PROGRAM P3_05_BatchTrail
VAR
	stDBParam 					:ST_BatchTrail;	
	fbDBWrite					:FB_PLCDBWriteEvt(sNetId:=CONST.AMS_NETID, tTimeout:=DEFAULT_ADS_TIMEOUT);
	tableColumns				:ARRAY [0..5] OF STRING(50) := ['batch', 'event', 'description', 'user', 'oldvalue', 'newvalue'];
	arrParam					:ARRAY [0..5] OF ST_ExpParameter := [(sParaName := 'batch', nParaSize := 101, eParaType := E_EXPPARAMETERTYPE.STRING_),
															 (sParaName := 'event', nParaSize := 101, eParaType := E_EXPPARAMETERTYPE.STRING_),
															 (sParaName := 'description', nParaSize := 101, eParaType := E_EXPPARAMETERTYPE.STRING_),
															 (sParaName := 'user', nParaSize := 101, eParaType := E_EXPPARAMETERTYPE.STRING_),
															 (sParaName := 'oldvalue', nParaSize := 101, eParaType := E_EXPPARAMETERTYPE.STRING_),
															 (sParaName := 'newvalue', nParaSize := 101, eParaType := E_EXPPARAMETERTYPE.STRING_)];
	fbDeleteTable    			:FB_PLCDBCmdEvt(sNetID:=CONST.AMS_NETID, tTimeout:=DEFAULT_ADS_TIMEOUT);
	fbBatchTrailWrite			:ARRAY[0..70] OF FB_AuditTrail_Write;
	sDeleteBatch				:STRING;	
	sDeleteAll					:STRING;
	sDelete						:STRING;
	bDelete						:BOOL;								
	bWrite						:BOOL;
	
	sProdCurrentPhase			:STRING;
	sCleanCurrentPhase			:STRING;
END_VAR
VAR // added by the converter: edge detectors and wires of the graphical bodies
    _rt1 : R_TRIG;
END_VAR

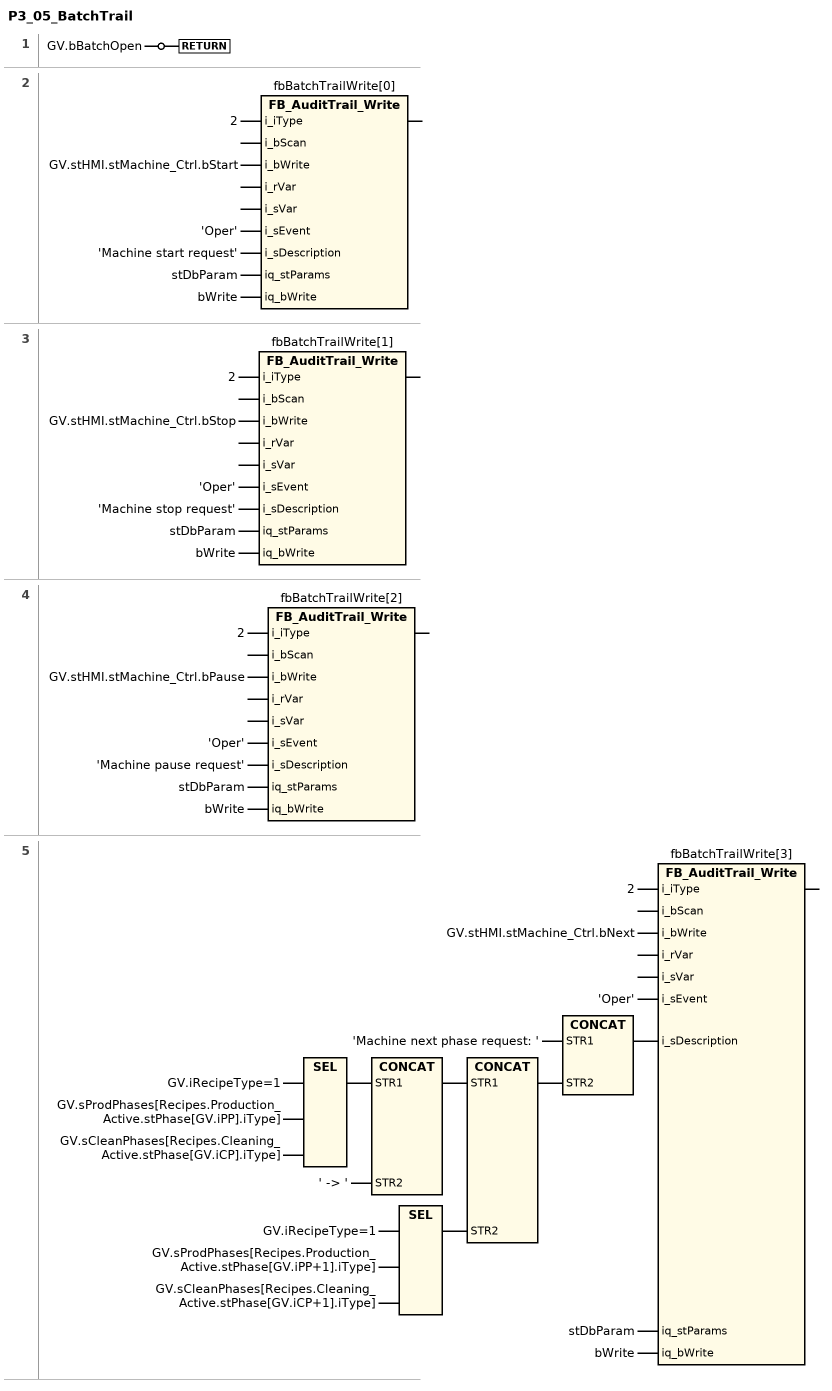
// NETWORK 1
IF NOT GV.bBatchOpen THEN RETURN; END_IF

// NETWORK 2
fbBatchTrailWrite[0](
    i_iType := 2,
    i_bWrite := GV.stHMI.stMachine_Ctrl.bStart,
    i_sEvent := 'Oper',
    i_sDescription := 'Machine start request',
    iq_stParams := stDbParam,
    iq_bWrite := bWrite); // FB_AuditTrail_Write

// NETWORK 3
fbBatchTrailWrite[1](
    i_iType := 2,
    i_bWrite := GV.stHMI.stMachine_Ctrl.bStop,
    i_sEvent := 'Oper',
    i_sDescription := 'Machine stop request',
    iq_stParams := stDbParam,
    iq_bWrite := bWrite); // FB_AuditTrail_Write

// NETWORK 4
fbBatchTrailWrite[2](
    i_iType := 2,
    i_bWrite := GV.stHMI.stMachine_Ctrl.bPause,
    i_sEvent := 'Oper',
    i_sDescription := 'Machine pause request',
    iq_stParams := stDbParam,
    iq_bWrite := bWrite); // FB_AuditTrail_Write

// NETWORK 5
fbBatchTrailWrite[3](
    i_iType := 2,
    i_bWrite := GV.stHMI.stMachine_Ctrl.bNext,
    i_sEvent := 'Oper',
    i_sDescription := CONCAT(STR1 := 'Machine next phase request: ', STR2 := CONCAT(STR1 := CONCAT(STR1 := SEL(GV.iRecipeType=1, GV.sProdPhases[Recipes.Production_Active.stPhase[GV.iPP].iType], GV.sCleanPhases[Recipes.Cleaning_Active.stPhase[GV.iCP].iType]), STR2 := ' -> '), STR2 := SEL(GV.iRecipeType=1, GV.sProdPhases[Recipes.Production_Active.stPhase[GV.iPP+1].iType], GV.sCleanPhases[Recipes.Cleaning_Active.stPhase[GV.iCP+1].iType]))),
    iq_stParams := stDbParam,
    iq_bWrite := bWrite); // FB_AuditTrail_Write

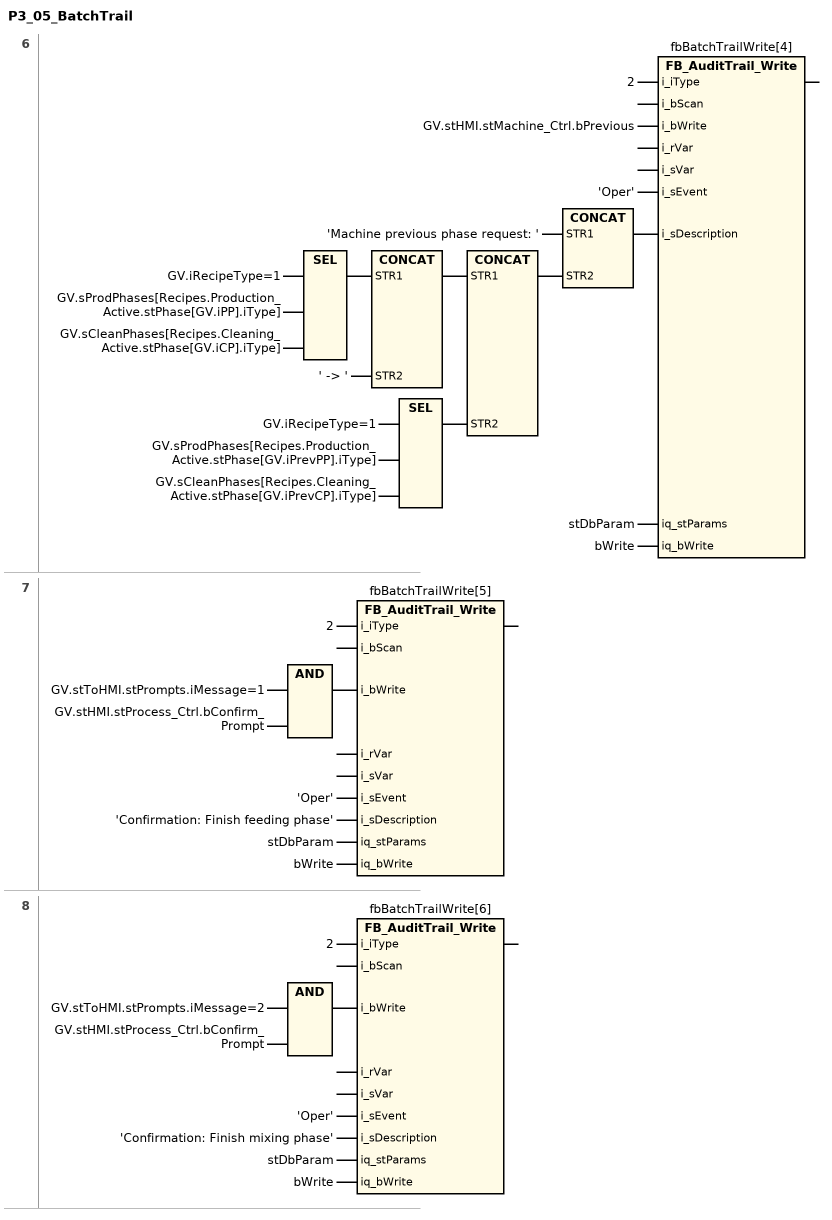
// NETWORK 6
fbBatchTrailWrite[4](
    i_iType := 2,
    i_bWrite := GV.stHMI.stMachine_Ctrl.bPrevious,
    i_sEvent := 'Oper',
    i_sDescription := CONCAT(STR1 := 'Machine previous phase request: ', STR2 := CONCAT(STR1 := CONCAT(STR1 := SEL(GV.iRecipeType=1, GV.sProdPhases[Recipes.Production_Active.stPhase[GV.iPP].iType], GV.sCleanPhases[Recipes.Cleaning_Active.stPhase[GV.iCP].iType]), STR2 := ' -> '), STR2 := SEL(GV.iRecipeType=1, GV.sProdPhases[Recipes.Production_Active.stPhase[GV.iPrevPP].iType], GV.sCleanPhases[Recipes.Cleaning_Active.stPhase[GV.iPrevCP].iType]))),
    iq_stParams := stDbParam,
    iq_bWrite := bWrite); // FB_AuditTrail_Write

// NETWORK 7
fbBatchTrailWrite[5](
    i_iType := 2,
    i_bWrite := (GV.stToHMI.stPrompts.iMessage=1) AND GV.stHMI.stProcess_Ctrl.bConfirm_Prompt,
    i_sEvent := 'Oper',
    i_sDescription := 'Confirmation: Finish feeding phase',
    iq_stParams := stDbParam,
    iq_bWrite := bWrite); // FB_AuditTrail_Write

// NETWORK 8
fbBatchTrailWrite[6](
    i_iType := 2,
    i_bWrite := (GV.stToHMI.stPrompts.iMessage=2) AND GV.stHMI.stProcess_Ctrl.bConfirm_Prompt,
    i_sEvent := 'Oper',
    i_sDescription := 'Confirmation: Finish mixing phase',
    iq_stParams := stDbParam,
    iq_bWrite := bWrite); // FB_AuditTrail_Write

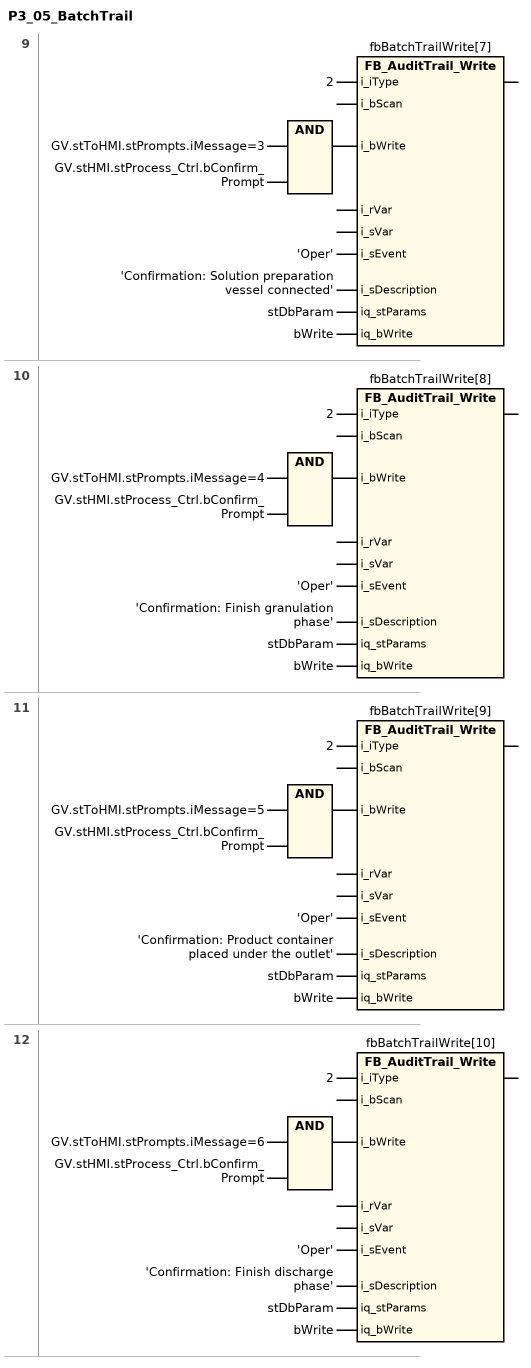
// NETWORK 9
fbBatchTrailWrite[7](
    i_iType := 2,
    i_bWrite := (GV.stToHMI.stPrompts.iMessage=3) AND GV.stHMI.stProcess_Ctrl.bConfirm_Prompt,
    i_sEvent := 'Oper',
    i_sDescription := 'Confirmation: Solution preparation vessel connected',
    iq_stParams := stDbParam,
    iq_bWrite := bWrite); // FB_AuditTrail_Write

// NETWORK 10
fbBatchTrailWrite[8](
    i_iType := 2,
    i_bWrite := (GV.stToHMI.stPrompts.iMessage=4) AND GV.stHMI.stProcess_Ctrl.bConfirm_Prompt,
    i_sEvent := 'Oper',
    i_sDescription := 'Confirmation: Finish granulation phase',
    iq_stParams := stDbParam,
    iq_bWrite := bWrite); // FB_AuditTrail_Write

// NETWORK 11
fbBatchTrailWrite[9](
    i_iType := 2,
    i_bWrite := (GV.stToHMI.stPrompts.iMessage=5) AND GV.stHMI.stProcess_Ctrl.bConfirm_Prompt,
    i_sEvent := 'Oper',
    i_sDescription := 'Confirmation: Product container placed under the outlet',
    iq_stParams := stDbParam,
    iq_bWrite := bWrite); // FB_AuditTrail_Write

// NETWORK 12
fbBatchTrailWrite[10](
    i_iType := 2,
    i_bWrite := (GV.stToHMI.stPrompts.iMessage=6) AND GV.stHMI.stProcess_Ctrl.bConfirm_Prompt,
    i_sEvent := 'Oper',
    i_sDescription := 'Confirmation: Finish discharge phase',
    iq_stParams := stDbParam,
    iq_bWrite := bWrite); // FB_AuditTrail_Write

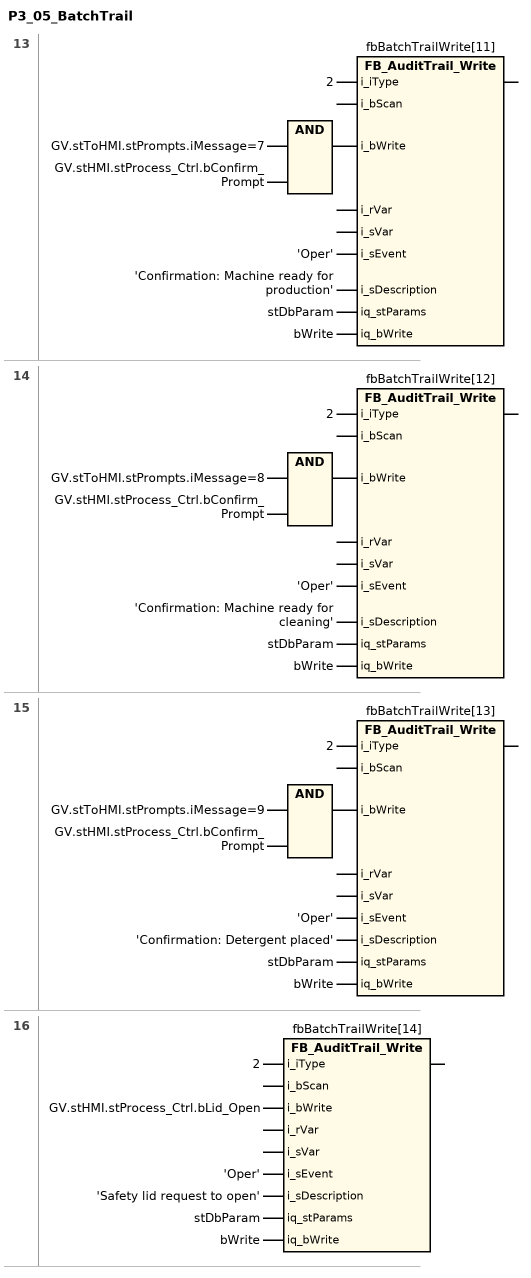
// NETWORK 13
fbBatchTrailWrite[11](
    i_iType := 2,
    i_bWrite := (GV.stToHMI.stPrompts.iMessage=7) AND GV.stHMI.stProcess_Ctrl.bConfirm_Prompt,
    i_sEvent := 'Oper',
    i_sDescription := 'Confirmation: Machine ready for production',
    iq_stParams := stDbParam,
    iq_bWrite := bWrite); // FB_AuditTrail_Write

// NETWORK 14
fbBatchTrailWrite[12](
    i_iType := 2,
    i_bWrite := (GV.stToHMI.stPrompts.iMessage=8) AND GV.stHMI.stProcess_Ctrl.bConfirm_Prompt,
    i_sEvent := 'Oper',
    i_sDescription := 'Confirmation: Machine ready for cleaning',
    iq_stParams := stDbParam,
    iq_bWrite := bWrite); // FB_AuditTrail_Write

// NETWORK 15
fbBatchTrailWrite[13](
    i_iType := 2,
    i_bWrite := (GV.stToHMI.stPrompts.iMessage=9) AND GV.stHMI.stProcess_Ctrl.bConfirm_Prompt,
    i_sEvent := 'Oper',
    i_sDescription := 'Confirmation: Detergent placed',
    iq_stParams := stDbParam,
    iq_bWrite := bWrite); // FB_AuditTrail_Write

// NETWORK 16
fbBatchTrailWrite[14](
    i_iType := 2,
    i_bWrite := GV.stHMI.stProcess_Ctrl.bLid_Open,
    i_sEvent := 'Oper',
    i_sDescription := 'Safety lid request to open',
    iq_stParams := stDbParam,
    iq_bWrite := bWrite); // FB_AuditTrail_Write

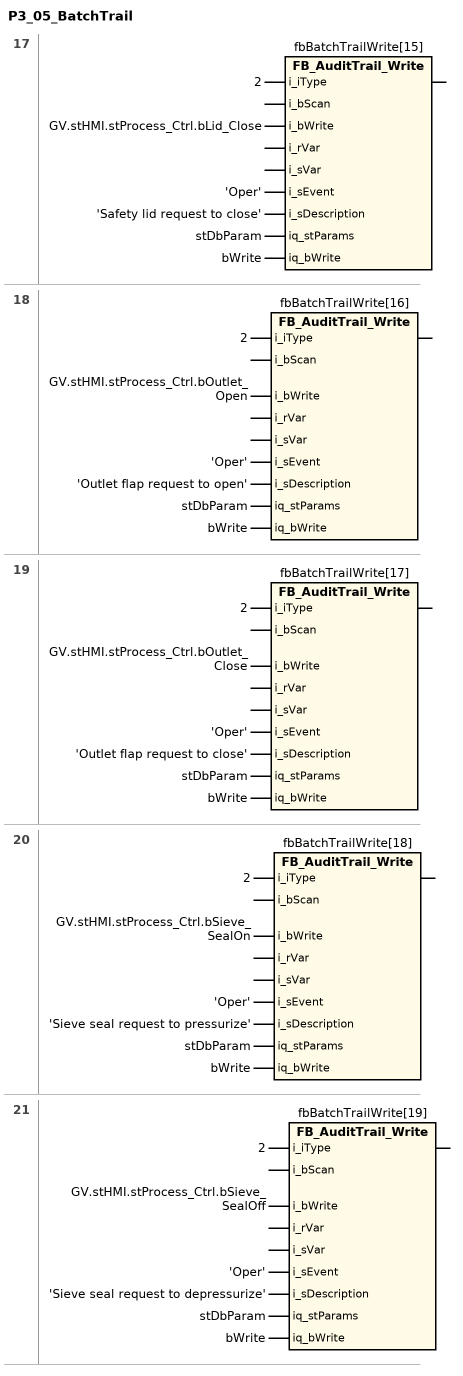
// NETWORK 17
fbBatchTrailWrite[15](
    i_iType := 2,
    i_bWrite := GV.stHMI.stProcess_Ctrl.bLid_Close,
    i_sEvent := 'Oper',
    i_sDescription := 'Safety lid request to close',
    iq_stParams := stDbParam,
    iq_bWrite := bWrite); // FB_AuditTrail_Write

// NETWORK 18
fbBatchTrailWrite[16](
    i_iType := 2,
    i_bWrite := GV.stHMI.stProcess_Ctrl.bOutlet_Open,
    i_sEvent := 'Oper',
    i_sDescription := 'Outlet flap request to open',
    iq_stParams := stDbParam,
    iq_bWrite := bWrite); // FB_AuditTrail_Write

// NETWORK 19
fbBatchTrailWrite[17](
    i_iType := 2,
    i_bWrite := GV.stHMI.stProcess_Ctrl.bOutlet_Close,
    i_sEvent := 'Oper',
    i_sDescription := 'Outlet flap request to close',
    iq_stParams := stDbParam,
    iq_bWrite := bWrite); // FB_AuditTrail_Write

// NETWORK 20
fbBatchTrailWrite[18](
    i_iType := 2,
    i_bWrite := GV.stHMI.stProcess_Ctrl.bSieve_SealOn,
    i_sEvent := 'Oper',
    i_sDescription := 'Sieve seal request to pressurize',
    iq_stParams := stDbParam,
    iq_bWrite := bWrite); // FB_AuditTrail_Write

// NETWORK 21
fbBatchTrailWrite[19](
    i_iType := 2,
    i_bWrite := GV.stHMI.stProcess_Ctrl.bSieve_SealOff,
    i_sEvent := 'Oper',
    i_sDescription := 'Sieve seal request to depressurize',
    iq_stParams := stDbParam,
    iq_bWrite := bWrite); // FB_AuditTrail_Write

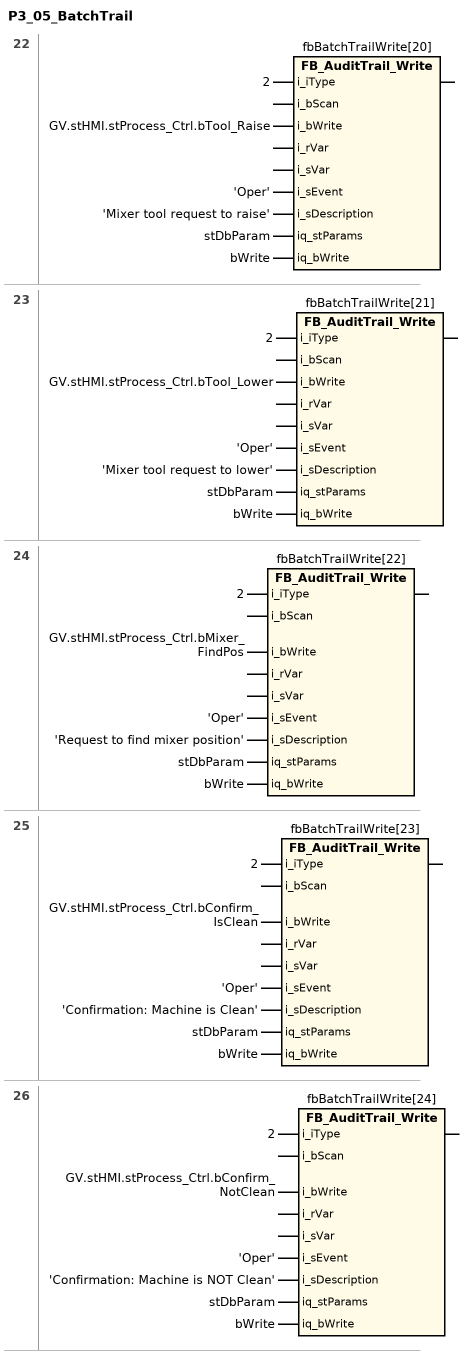
// NETWORK 22
fbBatchTrailWrite[20](
    i_iType := 2,
    i_bWrite := GV.stHMI.stProcess_Ctrl.bTool_Raise,
    i_sEvent := 'Oper',
    i_sDescription := 'Mixer tool request to raise',
    iq_stParams := stDbParam,
    iq_bWrite := bWrite); // FB_AuditTrail_Write

// NETWORK 23
fbBatchTrailWrite[21](
    i_iType := 2,
    i_bWrite := GV.stHMI.stProcess_Ctrl.bTool_Lower,
    i_sEvent := 'Oper',
    i_sDescription := 'Mixer tool request to lower',
    iq_stParams := stDbParam,
    iq_bWrite := bWrite); // FB_AuditTrail_Write

// NETWORK 24
fbBatchTrailWrite[22](
    i_iType := 2,
    i_bWrite := GV.stHMI.stProcess_Ctrl.bMixer_FindPos,
    i_sEvent := 'Oper',
    i_sDescription := 'Request to find mixer position',
    iq_stParams := stDbParam,
    iq_bWrite := bWrite); // FB_AuditTrail_Write

// NETWORK 25
fbBatchTrailWrite[23](
    i_iType := 2,
    i_bWrite := GV.stHMI.stProcess_Ctrl.bConfirm_IsClean,
    i_sEvent := 'Oper',
    i_sDescription := 'Confirmation: Machine is Clean',
    iq_stParams := stDbParam,
    iq_bWrite := bWrite); // FB_AuditTrail_Write

// NETWORK 26
fbBatchTrailWrite[24](
    i_iType := 2,
    i_bWrite := GV.stHMI.stProcess_Ctrl.bConfirm_NotClean,
    i_sEvent := 'Oper',
    i_sDescription := 'Confirmation: Machine is NOT Clean',
    iq_stParams := stDbParam,
    iq_bWrite := bWrite); // FB_AuditTrail_Write

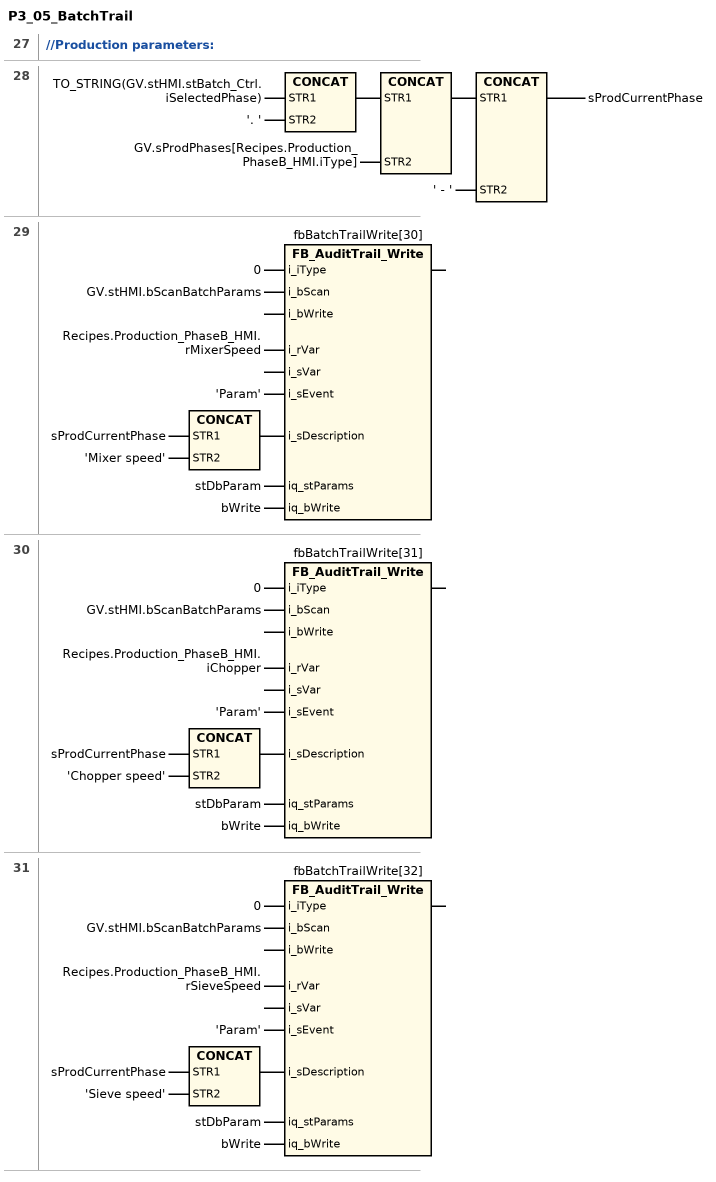
// NETWORK 27
// label: //Production parameters

// NETWORK 28
sProdCurrentPhase := CONCAT(STR1 := CONCAT(STR1 := CONCAT(STR1 := TO_STRING(GV.stHMI.stBatch_Ctrl.iSelectedPhase), STR2 := '. '), STR2 := GV.sProdPhases[Recipes.Production_PhaseB_HMI.iType]), STR2 := ' - ');

// NETWORK 29
fbBatchTrailWrite[30](
    i_iType := 0,
    i_bScan := GV.stHMI.bScanBatchParams,
    i_rVar := Recipes.Production_PhaseB_HMI.rMixerSpeed,
    i_sEvent := 'Param',
    i_sDescription := CONCAT(STR1 := sProdCurrentPhase, STR2 := 'Mixer speed'),
    iq_stParams := stDbParam,
    iq_bWrite := bWrite); // FB_AuditTrail_Write

// NETWORK 30
fbBatchTrailWrite[31](
    i_iType := 0,
    i_bScan := GV.stHMI.bScanBatchParams,
    i_rVar := Recipes.Production_PhaseB_HMI.iChopper,
    i_sEvent := 'Param',
    i_sDescription := CONCAT(STR1 := sProdCurrentPhase, STR2 := 'Chopper speed'),
    iq_stParams := stDbParam,
    iq_bWrite := bWrite); // FB_AuditTrail_Write

// NETWORK 31
fbBatchTrailWrite[32](
    i_iType := 0,
    i_bScan := GV.stHMI.bScanBatchParams,
    i_rVar := Recipes.Production_PhaseB_HMI.rSieveSpeed,
    i_sEvent := 'Param',
    i_sDescription := CONCAT(STR1 := sProdCurrentPhase, STR2 := 'Sieve speed'),
    iq_stParams := stDbParam,
    iq_bWrite := bWrite); // FB_AuditTrail_Write

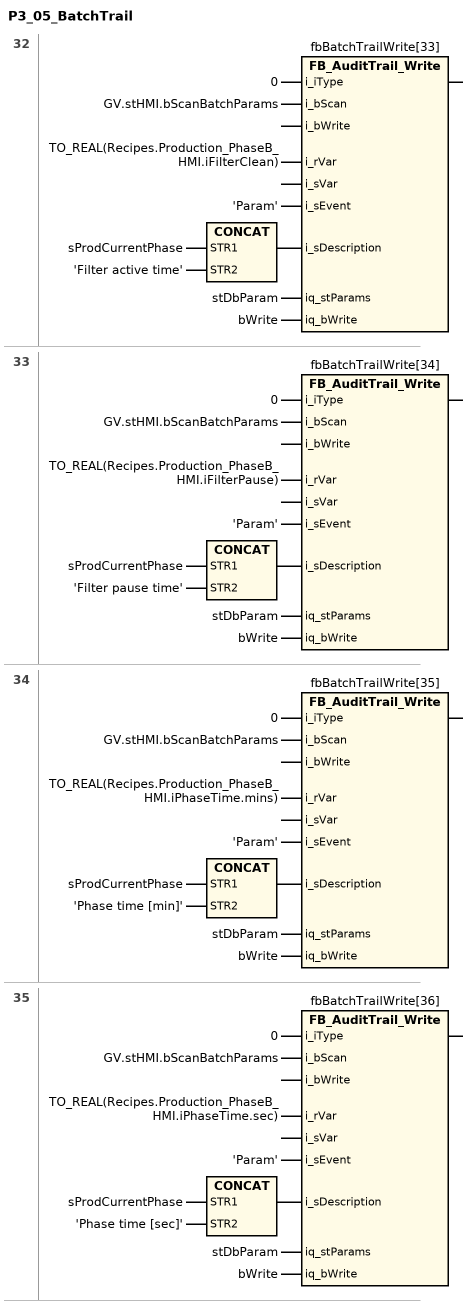
// NETWORK 32
fbBatchTrailWrite[33](
    i_iType := 0,
    i_bScan := GV.stHMI.bScanBatchParams,
    i_rVar := TO_REAL(Recipes.Production_PhaseB_HMI.iFilterClean),
    i_sEvent := 'Param',
    i_sDescription := CONCAT(STR1 := sProdCurrentPhase, STR2 := 'Filter active time'),
    iq_stParams := stDbParam,
    iq_bWrite := bWrite); // FB_AuditTrail_Write

// NETWORK 33
fbBatchTrailWrite[34](
    i_iType := 0,
    i_bScan := GV.stHMI.bScanBatchParams,
    i_rVar := TO_REAL(Recipes.Production_PhaseB_HMI.iFilterPause),
    i_sEvent := 'Param',
    i_sDescription := CONCAT(STR1 := sProdCurrentPhase, STR2 := 'Filter pause time'),
    iq_stParams := stDbParam,
    iq_bWrite := bWrite); // FB_AuditTrail_Write

// NETWORK 34
fbBatchTrailWrite[35](
    i_iType := 0,
    i_bScan := GV.stHMI.bScanBatchParams,
    i_rVar := TO_REAL(Recipes.Production_PhaseB_HMI.iPhaseTime.mins),
    i_sEvent := 'Param',
    i_sDescription := CONCAT(STR1 := sProdCurrentPhase, STR2 := 'Phase time [min]'),
    iq_stParams := stDbParam,
    iq_bWrite := bWrite); // FB_AuditTrail_Write

// NETWORK 35
fbBatchTrailWrite[36](
    i_iType := 0,
    i_bScan := GV.stHMI.bScanBatchParams,
    i_rVar := TO_REAL(Recipes.Production_PhaseB_HMI.iPhaseTime.sec),
    i_sEvent := 'Param',
    i_sDescription := CONCAT(STR1 := sProdCurrentPhase, STR2 := 'Phase time [sec]'),
    iq_stParams := stDbParam,
    iq_bWrite := bWrite); // FB_AuditTrail_Write

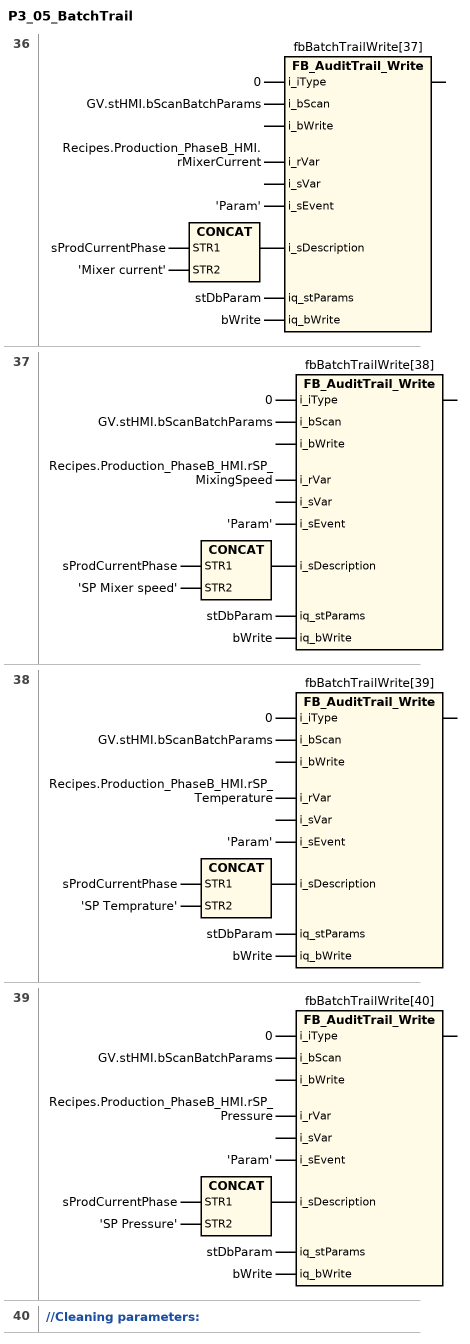
// NETWORK 36
fbBatchTrailWrite[37](
    i_iType := 0,
    i_bScan := GV.stHMI.bScanBatchParams,
    i_rVar := Recipes.Production_PhaseB_HMI.rMixerCurrent,
    i_sEvent := 'Param',
    i_sDescription := CONCAT(STR1 := sProdCurrentPhase, STR2 := 'Mixer current'),
    iq_stParams := stDbParam,
    iq_bWrite := bWrite); // FB_AuditTrail_Write

// NETWORK 37
fbBatchTrailWrite[38](
    i_iType := 0,
    i_bScan := GV.stHMI.bScanBatchParams,
    i_rVar := Recipes.Production_PhaseB_HMI.rSP_MixingSpeed,
    i_sEvent := 'Param',
    i_sDescription := CONCAT(STR1 := sProdCurrentPhase, STR2 := 'SP Mixer speed'),
    iq_stParams := stDbParam,
    iq_bWrite := bWrite); // FB_AuditTrail_Write

// NETWORK 38
fbBatchTrailWrite[39](
    i_iType := 0,
    i_bScan := GV.stHMI.bScanBatchParams,
    i_rVar := Recipes.Production_PhaseB_HMI.rSP_Temperature,
    i_sEvent := 'Param',
    i_sDescription := CONCAT(STR1 := sProdCurrentPhase, STR2 := 'SP Temprature'),
    iq_stParams := stDbParam,
    iq_bWrite := bWrite); // FB_AuditTrail_Write

// NETWORK 39
fbBatchTrailWrite[40](
    i_iType := 0,
    i_bScan := GV.stHMI.bScanBatchParams,
    i_rVar := Recipes.Production_PhaseB_HMI.rSP_Pressure,
    i_sEvent := 'Param',
    i_sDescription := CONCAT(STR1 := sProdCurrentPhase, STR2 := 'SP Pressure'),
    iq_stParams := stDbParam,
    iq_bWrite := bWrite); // FB_AuditTrail_Write

// NETWORK 40
// label: //Cleaning parameters

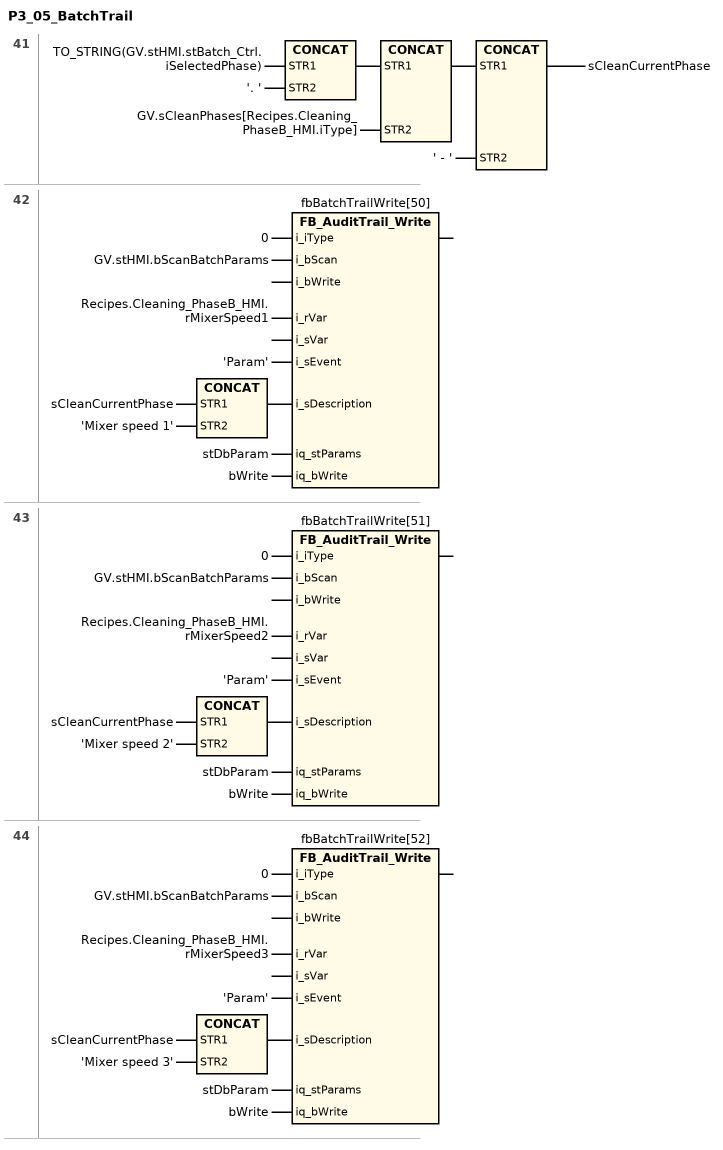
// NETWORK 41
sCleanCurrentPhase := CONCAT(STR1 := CONCAT(STR1 := CONCAT(STR1 := TO_STRING(GV.stHMI.stBatch_Ctrl.iSelectedPhase), STR2 := '. '), STR2 := GV.sCleanPhases[Recipes.Cleaning_PhaseB_HMI.iType]), STR2 := ' - ');

// NETWORK 42
fbBatchTrailWrite[50](
    i_iType := 0,
    i_bScan := GV.stHMI.bScanBatchParams,
    i_rVar := Recipes.Cleaning_PhaseB_HMI.rMixerSpeed1,
    i_sEvent := 'Param',
    i_sDescription := CONCAT(STR1 := sCleanCurrentPhase, STR2 := 'Mixer speed 1'),
    iq_stParams := stDbParam,
    iq_bWrite := bWrite); // FB_AuditTrail_Write

// NETWORK 43
fbBatchTrailWrite[51](
    i_iType := 0,
    i_bScan := GV.stHMI.bScanBatchParams,
    i_rVar := Recipes.Cleaning_PhaseB_HMI.rMixerSpeed2,
    i_sEvent := 'Param',
    i_sDescription := CONCAT(STR1 := sCleanCurrentPhase, STR2 := 'Mixer speed 2'),
    iq_stParams := stDbParam,
    iq_bWrite := bWrite); // FB_AuditTrail_Write

// NETWORK 44
fbBatchTrailWrite[52](
    i_iType := 0,
    i_bScan := GV.stHMI.bScanBatchParams,
    i_rVar := Recipes.Cleaning_PhaseB_HMI.rMixerSpeed3,
    i_sEvent := 'Param',
    i_sDescription := CONCAT(STR1 := sCleanCurrentPhase, STR2 := 'Mixer speed 3'),
    iq_stParams := stDbParam,
    iq_bWrite := bWrite); // FB_AuditTrail_Write

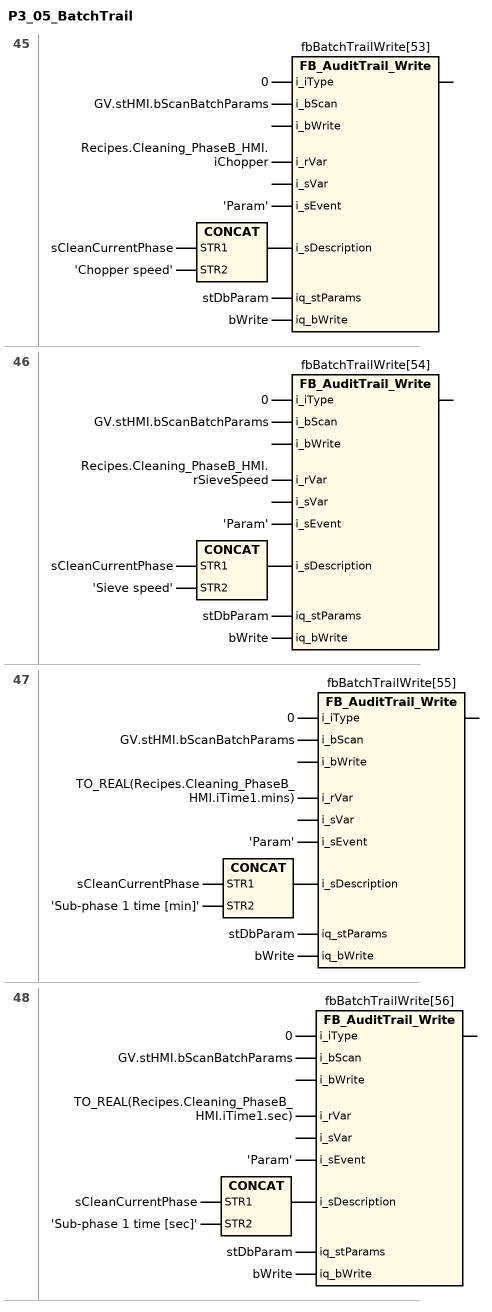
// NETWORK 45
fbBatchTrailWrite[53](
    i_iType := 0,
    i_bScan := GV.stHMI.bScanBatchParams,
    i_rVar := Recipes.Cleaning_PhaseB_HMI.iChopper,
    i_sEvent := 'Param',
    i_sDescription := CONCAT(STR1 := sCleanCurrentPhase, STR2 := 'Chopper speed'),
    iq_stParams := stDbParam,
    iq_bWrite := bWrite); // FB_AuditTrail_Write

// NETWORK 46
fbBatchTrailWrite[54](
    i_iType := 0,
    i_bScan := GV.stHMI.bScanBatchParams,
    i_rVar := Recipes.Cleaning_PhaseB_HMI.rSieveSpeed,
    i_sEvent := 'Param',
    i_sDescription := CONCAT(STR1 := sCleanCurrentPhase, STR2 := 'Sieve speed'),
    iq_stParams := stDbParam,
    iq_bWrite := bWrite); // FB_AuditTrail_Write

// NETWORK 47
fbBatchTrailWrite[55](
    i_iType := 0,
    i_bScan := GV.stHMI.bScanBatchParams,
    i_rVar := TO_REAL(Recipes.Cleaning_PhaseB_HMI.iTime1.mins),
    i_sEvent := 'Param',
    i_sDescription := CONCAT(STR1 := sCleanCurrentPhase, STR2 := 'Sub-phase 1 time [min]'),
    iq_stParams := stDbParam,
    iq_bWrite := bWrite); // FB_AuditTrail_Write

// NETWORK 48
fbBatchTrailWrite[56](
    i_iType := 0,
    i_bScan := GV.stHMI.bScanBatchParams,
    i_rVar := TO_REAL(Recipes.Cleaning_PhaseB_HMI.iTime1.sec),
    i_sEvent := 'Param',
    i_sDescription := CONCAT(STR1 := sCleanCurrentPhase, STR2 := 'Sub-phase 1 time [sec]'),
    iq_stParams := stDbParam,
    iq_bWrite := bWrite); // FB_AuditTrail_Write

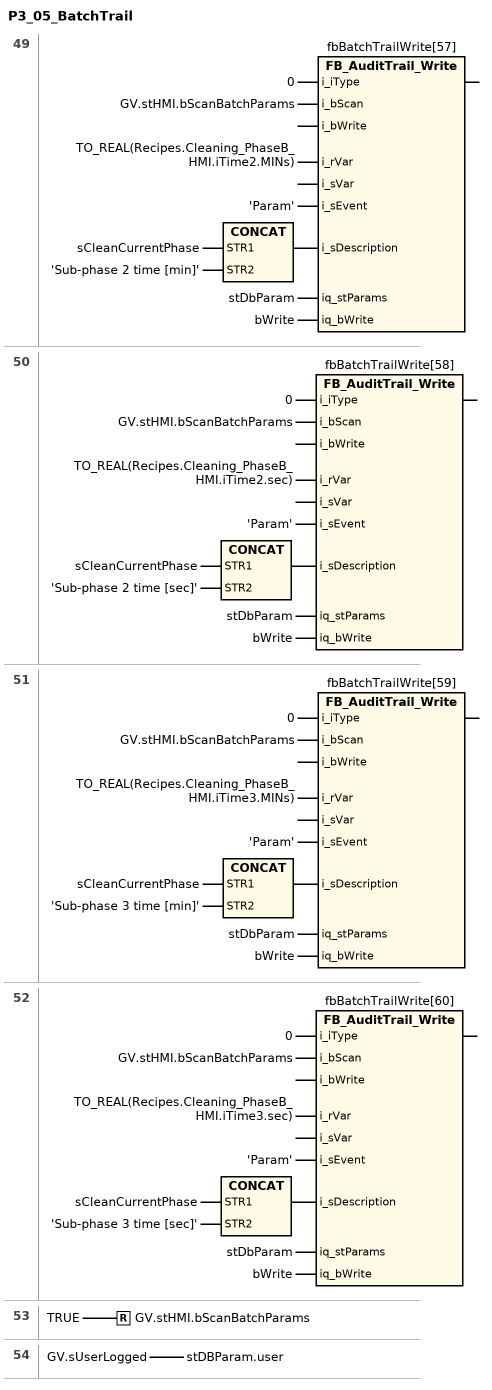
// NETWORK 49
fbBatchTrailWrite[57](
    i_iType := 0,
    i_bScan := GV.stHMI.bScanBatchParams,
    i_rVar := TO_REAL(Recipes.Cleaning_PhaseB_HMI.iTime2.MINs),
    i_sEvent := 'Param',
    i_sDescription := CONCAT(STR1 := sCleanCurrentPhase, STR2 := 'Sub-phase 2 time [min]'),
    iq_stParams := stDbParam,
    iq_bWrite := bWrite); // FB_AuditTrail_Write

// NETWORK 50
fbBatchTrailWrite[58](
    i_iType := 0,
    i_bScan := GV.stHMI.bScanBatchParams,
    i_rVar := TO_REAL(Recipes.Cleaning_PhaseB_HMI.iTime2.sec),
    i_sEvent := 'Param',
    i_sDescription := CONCAT(STR1 := sCleanCurrentPhase, STR2 := 'Sub-phase 2 time [sec]'),
    iq_stParams := stDbParam,
    iq_bWrite := bWrite); // FB_AuditTrail_Write

// NETWORK 51
fbBatchTrailWrite[59](
    i_iType := 0,
    i_bScan := GV.stHMI.bScanBatchParams,
    i_rVar := TO_REAL(Recipes.Cleaning_PhaseB_HMI.iTime3.MINs),
    i_sEvent := 'Param',
    i_sDescription := CONCAT(STR1 := sCleanCurrentPhase, STR2 := 'Sub-phase 3 time [min]'),
    iq_stParams := stDbParam,
    iq_bWrite := bWrite); // FB_AuditTrail_Write

// NETWORK 52
fbBatchTrailWrite[60](
    i_iType := 0,
    i_bScan := GV.stHMI.bScanBatchParams,
    i_rVar := TO_REAL(Recipes.Cleaning_PhaseB_HMI.iTime3.sec),
    i_sEvent := 'Param',
    i_sDescription := CONCAT(STR1 := sCleanCurrentPhase, STR2 := 'Sub-phase 3 time [sec]'),
    iq_stParams := stDbParam,
    iq_bWrite := bWrite); // FB_AuditTrail_Write

// NETWORK 53
GV.stHMI.bScanBatchParams R= TRUE;

// NETWORK 54
stDBParam.user := GV.sUserLogged;

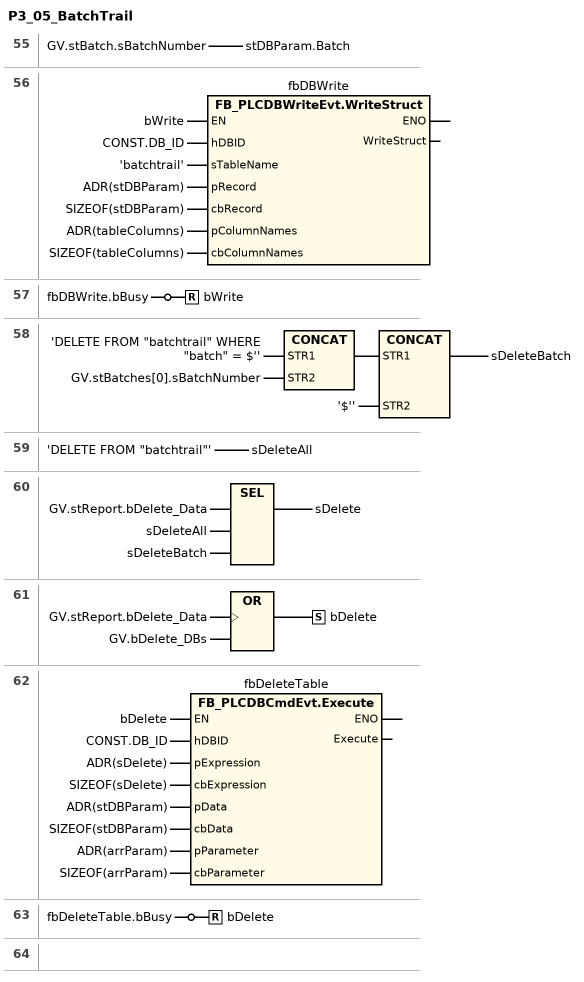
// NETWORK 55
stDBParam.Batch := GV.stBatch.sBatchNumber;

// NETWORK 56
IF bWrite THEN
    fbDBWrite.WriteStruct(
        hDBID := CONST.DB_ID,
        sTableName := 'batchtrail',
        pRecord := ADR(stDBParam),
        cbRecord := SIZEOF(stDBParam),
        pColumnNames := ADR(tableColumns),
        cbColumnNames := SIZEOF(tableColumns));
END_IF

// NETWORK 57
bWrite R= NOT fbDBWrite.bBusy;

// NETWORK 58
sDeleteBatch := CONCAT(STR1 := CONCAT(STR1 := 'DELETE FROM "batchtrail" WHERE "batch" = $'', STR2 := GV.stBatches[0].sBatchNumber), STR2 := '$'');

// NETWORK 59
sDeleteAll := 'DELETE FROM "batchtrail"';

// NETWORK 60
sDelete := SEL(GV.stReport.bDelete_Data, sDeleteAll, sDeleteBatch);

// NETWORK 61
_rt1(CLK := GV.stReport.bDelete_Data);
bDelete S= _rt1.Q OR GV.bDelete_DBs;

// NETWORK 62
IF bDelete THEN
    fbDeleteTable.Execute(
        hDBID := CONST.DB_ID,
        pExpression := ADR(sDelete),
        cbExpression := SIZEOF(sDelete),
        pData := ADR(stDBParam),
        cbData := SIZEOF(stDBParam),
        pParameter := ADR(arrParam),
        cbParameter := SIZEOF(arrParam));
END_IF

// NETWORK 63
bDelete R= NOT fbDeleteTable.bBusy;

// NETWORK 64

END_PROGRAM

(* stored: Version 1.1.0.1, ProductVersion 3.1.4026.13
   POU P3_05_BatchTrail: Id {f9aa9a80-3fc4-43b4-9583-d852c8f3be20}, SpecialFunc None *)
